Staubli VAL3: Prefix.dtx

mdesc mNomSpeed
public num nLength
